FUNCTION_BLOCK Copy of L3_CompletedPartHDLR_old_multi (* Basic Function Block Type *)
  (* Standard: 61499-2 *)
  (* Version 0.0, 2014-11-04, EQUEROL, UJI *)
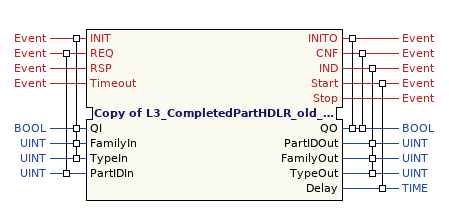
  EVENT_INPUT
    INIT WITH QI, FamilyIn, TypeIn; (* Initialization Request *)
    REQ WITH PartIDIn; (* Normal Execution Request *)
    RSP; (* Response from OrderManager *)
    Timeout; (* Timeout *)
  END_EVENT
  EVENT_OUTPUT
    INITO WITH QO; (* Initialization Confirm *)
    CNF WITH QO; (* Execution Confirmation *)
    IND WITH PartIDOut, FamilyOut, TypeOut; (* Indication to the OrderManager *)
    Start WITH Delay; (* Timeout start *)
    Stop; (* Timeout stop *)
  END_EVENT
  VAR_INPUT
    QI : BOOL; (* Input event qualifier *)
    FamilyIn : UINT; (* PP Family *)
    TypeIn : UINT; (* PP type *)
    PartIDIn : UINT; (* Completed part identifier *)
  END_VAR
  VAR_OUTPUT
    QO : BOOL; (* Output event qualifier *)
    PartIDOut : UINT; (* Part identifier *)
    FamilyOut : UINT; (* PP family *)
    TypeOut : UINT; (* PP type *)
    Delay : TIME; (* Timeout delay *)
  END_VAR
  VAR
    PartBuffer : ARRAY [0..9] OF UINT := [0,0,0,0,0,0,0,0,0,0]; (* Buffer holding completed parts *)
    BufferSize : USINT := 10; (* Buffer size *)
    HeadIndex : USINT := 0; (* Pointer to the head of the buffer *)
    TailIndex : USINT := 0; (* Pointer to the end of the buffer *)
    LastPart : BOOL := false; (* Variable indicating if the last part was received *)
  END_VAR
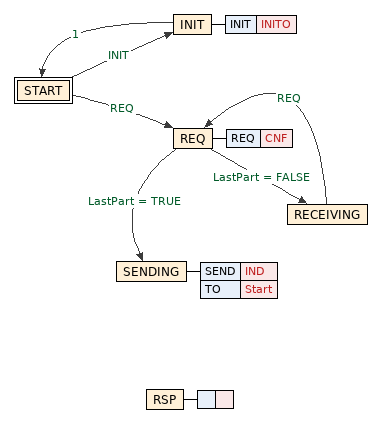
  EC_STATES
    START; (* Initial State *)
    INIT : INIT -> INITO; (* Initialization *)
    REQ : REQ -> CNF; (* Normal execution *)
    RECEIVING;
    SENDING : SEND -> IND, TO -> Start;
    RSP;
  END_STATES
  EC_TRANSITIONS
    START TO INIT := INIT;
    INIT TO START := 1;
    START TO REQ := REQ;
    REQ TO RECEIVING := LastPart = FALSE;
    REQ TO SENDING := LastPart = TRUE;
    RECEIVING TO REQ := REQ;
  END_TRANSITIONS
  ALGORITHM INIT IN ST: (* Initialization algorithm *)

  END_ALGORITHM
  ALGORITHM REQ IN ST: (* Normally executed algorithm *)
IF PartIDIn <> 0 THEN
	LastPart := FALSE;
	(*Stack the received order*)
	PartBuffer[HeadIndex] := PartIDIn;

	(*PostIncrement HeadIndex*)
	HeadIndex := HeadIndex + 1;
	IF HeadIndex >= BufferSize THEN
		HeadIndex := 0;
	END_IF;

	(*Check if buffer is full*)
	IF HeadIndex = TailIndex THEN
		(*Buffer is full, HeadIndex can't be incremented*)
		IF HeadIndex = 0 THEN
			HeadIndex := BufferSize - 1;
		ELSE
			HeadIndex := HeadIndex - 1;
		END_IF;
	END_IF;
ELSE
	(*Last part received, start sending to order manager*)
	LastPart := TRUE;
END_IF;
  END_ALGORITHM
  ALGORITHM RSP IN ST: (* new algorithm *)
(*Part correctly send*)
(*Increase tail index*)
TailIndex := TailIndex + 1;
IF TailIndex >= BufferSize THEN
	TailIndex := 0;
END_IF;
IF TailIndex = HeadIndex THEN
	LastPart := TRUE;
ELSE
	LastPart := FALSE;
END_IF;
  END_ALGORITHM
  ALGORITHM SEND IN ST: (* send algo *)
PartIDOut := PartBuffer[TailIndex];
FamilyOut := FamilyIn;
TypeOut := TypeIn;
  END_ALGORITHM
  ALGORITHM TO IN ST: (* TimeOut algo *)
Delay := TIME#1000ms;
  END_ALGORITHM
END_FUNCTION_BLOCK
